SUBAPPLICATION AR_S_TO_ATM (* Wandelt einen AR-Wert (REAL, Sekunden) in einen ATM-Wert (TIME) um - fuer TIME-Sockets (z.B. FT_PT1_AR.TM), die von einer per VT/Web einstellbaren, in Sekunden editierten REAL-Groesse (AR2) gespeist werden sollen. T#1s * Sekunden (adapter::iec61131::arithmetic::AR_MULTIME) - echte IEC-61131-3-TIME-Arithmetik, analog dem bereits bestehenden Sec_To_Time in INI_OPC_PARAM_ATM.SUB. *)
  (* Standard: 61499-2; Description: Copyright (c) 2026 Meisterschulen am Ostbahnhof This program and the accompanying materials are made available under the terms of the Eclipse Public License 2.0 which is available at https://www.eclipse.org/legal/epl-2.0/ SPDX-License-Identifier: EPL-2.0 *)
  (* Version 1.1, 2026-09-23, Franz Höpfinger, Meisterschulen am Ostbahnhof, Korrektur: die bisherige Kette (AR_R_MUL x1000 -> AR_TO_ADI -> ADI_TO_ATM) beruhte auf einer nicht existierenden Funktion iec61131::conversion::F_DINT_TO_TIME (Franz: 'F_DINT_TO_TIME GIBT ES NICHT'). Ersetzt durch AR_MULTIME (T#1s * REAL-Sekunden), bereits real erprobtes Muster aus INI_OPC_PARAM_ATM.SUB. ADI_TO_ATM.fbt geloescht (war erfunden). *)
  (* Version 1.0, 2026-09-22, Franz Höpfinger, Meisterschulen am Ostbahnhof, initial implementation - fuer die einstellbare PT1-Filterzeit der Puls-Frequenz-Sensoren (logiBUS_PI_Raw_Publish_OPC), Franz: 'Kunde will die Filter Zeit ohnehin Einstellbar haben (die 2S)'. *)
  PACKAGE MyLib::sys;
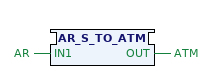
  SOCKETS
    IN1 : adapter::types::unidirectional::AR; (* Zeit in Sekunden (REAL) *)
  END_SOCKETS
  PLUGS
    OUT : adapter::types::unidirectional::ATM; (* IN1, umgerechnet von Sekunden (REAL) auf TIME *)
  END_PLUGS
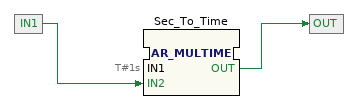
  FBS
    Sec_To_Time : adapter::iec61131::arithmetic::AR_MULTIME(IN1 := T#1s);
  END_FBS
  ADAPTER_CONNECTIONS
    IN1 TO Sec_To_Time.IN2;
    Sec_To_Time.OUT TO OUT;
  END_CONNECTIONS
END_SUBAPPLICATION
